(* CODESYS project Final_project.project

Project tree, tasks and I/O mapping:
  Device : CODESYS Control Win V3 x64, CODESYS, version 3.5.21.40
    application Application
      libraries: Standard, 3.5.18.0 (System); VisuDialogs, * (System)
      task MainTask (cyclic, interval t#20ms, priority 1) calls Step_0, Step_1, Step_2, Step_3
      task Faults (cyclic, interval t#20ms, priority 14) calls Faults
      task State_change (cyclic, interval t#20ms, priority 10) calls State_change
      task VISU_TASK (cyclic, interval 100 ms, priority 15) calls VisuElems.Visu_Prg
      program State_change [LD]
      program Step_0 [?]
      global variables GVL
      program Step_1 [?]
      program Step_2 [?]
      program Step_3 [?]
      program Faults [?]
      data type State
      visualisation HMI
    Modbus_COM : Modbus COM, CODESYS, version 4.4.0.0
        settings: DataBits = 8; StopBits = 1; ComPort = 1
      Modbus_Client_COM_Port : Modbus Client, COM Port, CODESYS, version 4.5.0.0
        Modbus_Server_COM_Port : Modbus Server, COM Port, CODESYS, version 4.5.0.0
            settings: Channel 0.Function Code = 2; Channel 0.Read Offset = 16#0000; Channel 0.Read Length = 10; Channel 0.Write Offset = 0; Channel 0.Write Length = 0; Channel 0.Cycle Time = 100; Channel 1.Function Code = 15; Channel 1.Read Offset = 0; Channel 1.Read Length = 0; Channel 1.Write Offset = 16#0000; Channel 1.Write Length = 8; Channel 1.Cycle Time = 100
            input  Application.GVL.Sprayer : BOOL  // Channel 0.Channel 0.Bit0
            input  Application.GVL.Squeegee : BOOL  // Channel 0.Channel 0.Bit1
            input  Application.GVL.Cloth : BOOL  // Channel 0.Channel 0.Bit2
            input  Application.GVL.PosMin : BOOL  // Channel 0.Channel 0.Bit3
            input  Application.GVL.PosMax : BOOL  // Channel 0.Channel 0.Bit4
            input  Application.GVL.Infrared : BOOL  // Channel 0.Channel 0.Bit5
            input  Application.GVL.RobotBit0 : BOOL  // Channel 0.Channel 0.Bit6
            input  Application.GVL.RobotBit1 : BOOL  // Channel 0.Channel 0.Bit7
            input  Application.GVL.RobotBit2 : BOOL  // Channel 0.Channel 0.Bit0
            input  Application.GVL.RobotBit3 : BOOL  // Channel 0.Channel 0.Bit1
            output Application.GVL.CmdBit0 : BOOL  // Channel 1.Channel 1.Bit2
            output Application.GVL.CmdBit1 : BOOL  // Channel 1.Channel 1.Bit3
            output Application.GVL.CmdBit2 : BOOL  // Channel 1.Channel 1.Bit4
            output Application.GVL.CmdBit3 : BOOL  // Channel 1.Channel 1.Bit5
            output Application.GVL.MotorCW : BOOL  // Channel 1.Channel 1.Bit6
            output Application.GVL.MotorCCW : BOOL  // Channel 1.Channel 1.Bit7
            unmapped channels: Channel 0, Channel 1
  text list GlobalTextList
*)

// Device/Application/State
TYPE State :
STRUCT
	isFaulted :BOOL;
	isRunning :BOOL;
	isStopped :BOOL;
	isPaused :BOOL;
END_STRUCT
END_TYPE

// Device/Application/GVL
{attribute 'qualified_only'}
VAR_GLOBAL
	StartBtn: BOOL;	  (*Start button*)
    StopBtn: BOOL;   (* Stop button *)
    Infrared: BOOL;   (* Obstacle sensor *)
	
    Sprayer     : BOOL;   (* Sprayer sensor *)
    Squeegee    : BOOL;   (* Squeegee sensor *)
    Cloth       : BOOL;   (* Cloth sensor *)
    PosMin: BOOL;
    PosMax      : BOOL;   (* Maximum position sensor *)

    RobotBit0   : BOOL;   (* Robot feedback bit 0 *)
    RobotBit1   : BOOL;   (* Robot feedback bit 1 *)
    RobotBit2   : BOOL;   (* Robot feedback bit 2 *)
    RobotBit3   : BOOL;   (* Robot feedback bit 3 *)

(*OUTPUTS*)
    CmdBit0     : BOOL;   (* 4-bit command to robot *)
    CmdBit1     : BOOL;
    CmdBit2     : BOOL;
    CmdBit3     : BOOL;

    MotorCW     : BOOL;   (* Motor moves up *)
    MotorCCW    : BOOL;   (* Motor moves down *)

(*internal memory *)
    STEP0       : BOOL;   (* go home(at max position)*)
    STEP1       : BOOL;   (* Task1: move down & spray *)
    STEP2       : BOOL;   (* Task2: now squeegee while moving up again *)
    STEP3       : BOOL;   (* Task3: cloth finishing and moving down again*)
	sprays_counter : CTU;
	Motor_timer :TON;
	reset_counter  : BOOL;
	check_water    : BOOL;
	cycle_finished : BOOL;
	one_shot       : R_TRIG;
	MSFault: BOOL;// Problem with the motor sensors
	SensorFault: BOOL;//problem with the tool sensors
	State : STATE;
	Reset_Faults :BOOL;
	Motor_Fault :BOOL; //Problem with the Motor
	Step2CTU : CTU;
	Step21 :BOOL; //substep 1 of step 2
	Step22 :BOOL; //substep 2 of step 2
	
END_VAR

// Device/Application/Step_0
PROGRAM Step_0
VAR
END_VAR

(* body of a kind this reader does not render *)

END_PROGRAM

// Device/Application/Step_1
PROGRAM Step_1
VAR
END_VAR

(* body of a kind this reader does not render *)

END_PROGRAM

// Device/Application/Step_2
PROGRAM Step_2
VAR
END_VAR

(* body of a kind this reader does not render *)

END_PROGRAM

// Device/Application/Step_3
PROGRAM Step_3
VAR
END_VAR

(* body of a kind this reader does not render *)

END_PROGRAM

// Device/Application/Faults
PROGRAM Faults
VAR
END_VAR

(* body of a kind this reader does not render *)

END_PROGRAM

// Device/Application/State_change
 PROGRAM State_change
VAR	
END_VAR
VAR // added by the converter: edge detectors and wires of the graphical bodies
    _w1, _w2, _w3 : BOOL;
END_VAR

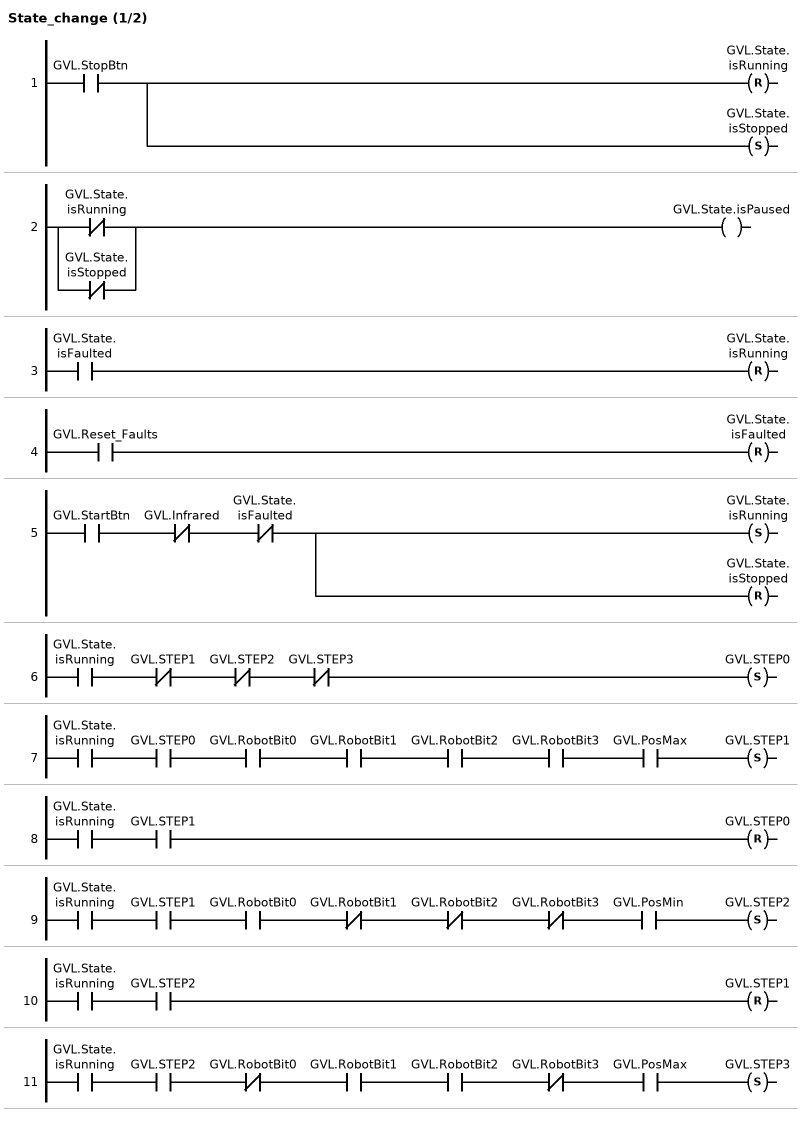
// NETWORK 1
_w1 := GVL.StopBtn;
GVL.State.isRunning R= _w1;
GVL.State.isStopped S= _w1;

// NETWORK 2
GVL.State.isPaused := NOT GVL.State.isRunning OR NOT GVL.State.isStopped;

// NETWORK 3
GVL.State.isRunning R= GVL.State.isFaulted;

// NETWORK 4
GVL.State.isFaulted R= GVL.Reset_Faults;

// NETWORK 5
_w2 := GVL.StartBtn AND NOT GVL.Infrared AND NOT GVL.State.isFaulted;
GVL.State.isRunning S= _w2;
GVL.State.isStopped R= _w2;

// NETWORK 6
GVL.STEP0 S= GVL.State.isRunning AND NOT GVL.STEP1 AND NOT GVL.STEP2 AND NOT GVL.STEP3;

// NETWORK 7
GVL.STEP1 S= GVL.State.isRunning AND GVL.STEP0 AND GVL.RobotBit0 AND GVL.RobotBit1 AND GVL.RobotBit2 AND GVL.RobotBit3 AND GVL.PosMax;

// NETWORK 8
GVL.STEP0 R= GVL.State.isRunning AND GVL.STEP1;

// NETWORK 9
GVL.STEP2 S= GVL.State.isRunning AND GVL.STEP1 AND GVL.RobotBit0 AND NOT GVL.RobotBit1 AND NOT GVL.RobotBit2 AND NOT GVL.RobotBit3 AND GVL.PosMin;

// NETWORK 10
GVL.STEP1 R= GVL.State.isRunning AND GVL.STEP2;

// NETWORK 11
GVL.STEP3 S= GVL.State.isRunning AND GVL.STEP2 AND NOT GVL.RobotBit0 AND GVL.RobotBit1 AND GVL.RobotBit2 AND NOT GVL.RobotBit3 AND GVL.PosMax;

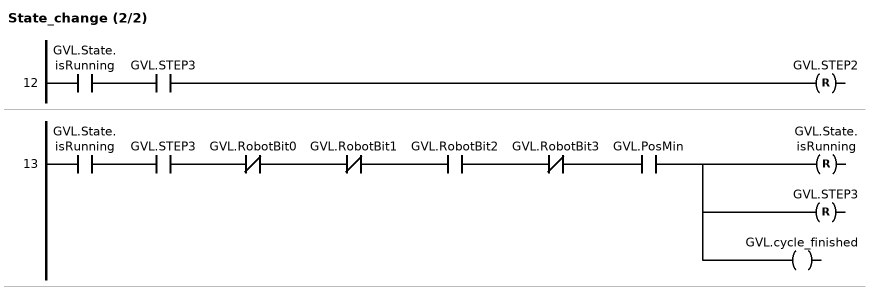
// NETWORK 12
GVL.STEP2 R= GVL.State.isRunning AND GVL.STEP3;

// NETWORK 13
_w3 := GVL.State.isRunning AND GVL.STEP3 AND NOT GVL.RobotBit0 AND NOT GVL.RobotBit1 AND GVL.RobotBit2 AND NOT GVL.RobotBit3 AND GVL.PosMin;
GVL.State.isRunning R= _w3;
GVL.STEP3 R= _w3;
GVL.cycle_finished := _w3;

END_PROGRAM

// Device/Application/HMI
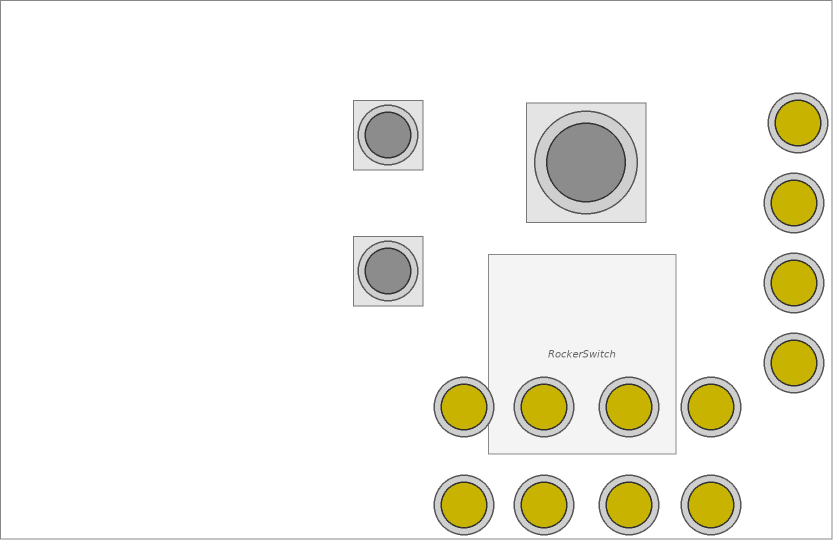
VISUALIZATION HMI  // 833x540
    Group (353,88 480x452)
        PushSwitch (0,12 70x70), behaviour: TOGGLE, style: Switch-PushSwitch-Gray
            OnValueChanged:  ToggleVariable=reset_counter
        PushSwitch (0,148 70x70), behaviour: TOGGLE, style: Switch-PushSwitch-Gray
            OnValueChanged:  ToggleVariable=Reset_Faults
        RockerSwitch (135,166 188x200), tooltip "Stop", behaviour: TOGGLE, style: Switch-RockerSwitch-Gray
            OnValueChanged:  ToggleVariable=STOP
        PushSwitch (173,13 120x123), tooltip "Start", variable: GVL.StartBtn, behaviour: TOGGLE, style: Switch-PushSwitch-Gray
            OnValueChanged:  ToggleVariable=StartBtn
        Lamp1 (410,0 70x70), variable: check_water, style: Lamp-Lamp1-Yellow
        Lamp1 (406,80 70x70), variable: MSFault, style: Lamp-Lamp1-Yellow
        Lamp1 (406,160 70x70), variable: SensorFault, style: Lamp-Lamp1-Yellow
        Lamp1 (406,240 70x70), variable: Motor_Fault, style: Lamp-Lamp1-Yellow
        Lamp1 (76,284 70x70), variable: State.isStopped, style: Lamp-Lamp1-Yellow
        Lamp1 (156,284 70x70), variable: State.isPaused, style: Lamp-Lamp1-Yellow
        Lamp1 (241,284 70x70), variable: State.isRunning, style: Lamp-Lamp1-Yellow
        Lamp1 (323,284 70x70), variable: State.isFaulted, style: Lamp-Lamp1-Yellow
        Lamp1 (76,382 70x70), variable: GVL.STEP0, style: Lamp-Lamp1-Yellow
        Lamp1 (156,382 70x70), variable: GVL.STEP1, style: Lamp-Lamp1-Yellow
        Lamp1 (241,382 70x70), variable: GVL.STEP2, style: Lamp-Lamp1-Yellow
        Lamp1 (323,382 70x70), variable: GVL.STEP3, style: Lamp-Lamp1-Yellow
END_VISUALIZATION
